FUNCTION_BLOCK FB_UML_SC
VAR
	// Transition condition
	bInitFinished				: BOOL;
	bUseXmlFormat				: BOOL;
	bAllInfoCopiedToFile		: BOOL;
	bSendToMasterFinished		: BOOL;
	bSendToClientFinished		: BOOL;
	
	// Counters
	nCounterInit				: INT;
	nCounterSaveInitSettings	: INT;
	nCounterClearXml			: INT;
	nCounterFillXml				: INT;
	nCounterSaveXml				: INT;
	nCounterClearText			: INT;
	nCounterFillText			: INT;
	nCounterSaveText			: INT;
	nCounterGetMasterID			: INT;
	nCounterGetClientID			: INT;
	nCounterSendToMaster		: INT;
	nCounterSendToClient		: INT;
	
	// Debugging
	bMasterFirst				: BOOL;
	bClientFirst				: BOOL;
END_VAR

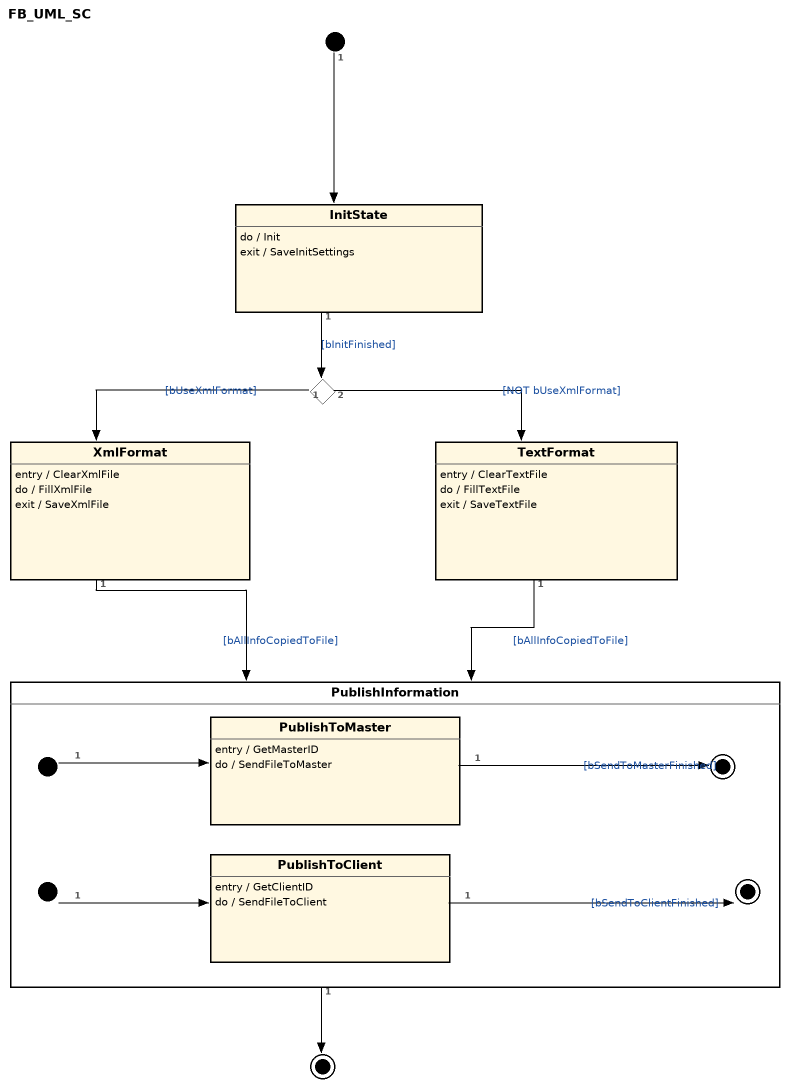
STATECHART FB_UML_SC  // abortable
    START StartState1
    STATE InitState
        do / Init
        exit / SaveInitSettings
    CHOICE ChoiceElement1
    STATE XmlFormat
        entry / ClearXmlFile
        do / FillXmlFile
        exit / SaveXmlFile
    STATE TextFormat
        entry / ClearTextFile
        do / FillTextFile
        exit / SaveTextFile
    COMPOSITE STATE PublishInformation
        REGION Region0 // priority 1
        START StartState2
        STATE PublishToMaster
            entry / GetMasterID
            do / SendFileToMaster
        END EndState2
        StartState2 -> PublishToMaster  // priority 1, on completion
        PublishToMaster -> EndState2 [bSendToMasterFinished] // priority 1
        REGION Region1 // priority 2
        START StartState3
        STATE PublishToClient
            entry / GetClientID
            do / SendFileToClient
        END EndState3
        StartState3 -> PublishToClient  // priority 1, on completion
        PublishToClient -> EndState3 [bSendToClientFinished] // priority 1
    END_STATE
    END EndState1
    StartState1 -> InitState  // priority 1, on completion
    InitState -> ChoiceElement1 [bInitFinished] // priority 1
    ChoiceElement1 -> XmlFormat [bUseXmlFormat] // priority 1
    ChoiceElement1 -> TextFormat [NOT bUseXmlFormat] // priority 2
    XmlFormat -> PublishInformation [bAllInfoCopiedToFile] // priority 1
    TextFormat -> PublishInformation [bAllInfoCopiedToFile] // priority 1
    PublishInformation -> EndState1  // priority 1, on completion
END_STATECHART

METHOD PROTECTED ClearTextFile
VAR_INPUT
END_VAR
nCounterClearText := nCounterClearText + 1;
END_METHOD

METHOD PROTECTED ClearXmlFile
VAR_INPUT
END_VAR
nCounterClearXml := nCounterClearXml + 1;
END_METHOD

METHOD PROTECTED FillTextFile
VAR_INPUT
END_VAR
nCounterFillText := nCounterFillText + 1;
END_METHOD

METHOD PROTECTED FillXmlFile
VAR_INPUT
END_VAR
nCounterFillXml := nCounterFillXml + 1;
END_METHOD

METHOD PROTECTED GetClientID
VAR_INPUT
END_VAR
nCounterGetClientID := nCounterGetClientID + 1;

IF NOT bMasterFirst THEN
	bClientFirst := TRUE;
END_IF
END_METHOD

METHOD PROTECTED GetMasterID
VAR_INPUT
END_VAR
nCounterGetMasterID := nCounterGetMasterID + 1;

IF NOT bClientFirst THEN
	bMasterFirst := TRUE;
END_IF
END_METHOD

METHOD PROTECTED Init
VAR_INPUT
END_VAR
nCounterInit := nCounterInit + 1;
END_METHOD

METHOD PROTECTED SaveInitSettings
VAR_INPUT
END_VAR
nCounterSaveInitSettings := nCounterSaveInitSettings + 1;

bInitFinished 			:= FALSE;
bAllInfoCopiedToFile 	:= FALSE;
bSendToClientFinished 	:= FALSE;
bSendToMasterFinished	:= FALSE;
bMasterFirst			:= FALSE;
bClientFirst			:= FALSE;
END_METHOD

METHOD PROTECTED SaveTextFile
VAR_INPUT
END_VAR
nCounterSaveText := nCounterSaveText + 1;
END_METHOD

METHOD PROTECTED SaveXmlFile
VAR_INPUT
END_VAR
nCounterSaveXml := nCounterSaveXml + 1;
END_METHOD

METHOD PROTECTED SendFileToClient
VAR_INPUT
END_VAR
nCounterSendToClient := nCounterSendToClient + 1;
END_METHOD

METHOD PROTECTED SendFileToMaster
VAR_INPUT
END_VAR
nCounterSendToMaster := nCounterSendToMaster + 1;
END_METHOD

END_FUNCTION_BLOCK

(* stored: Version 1.1.0.1, ProductVersion 3.1.4024.12
   POU FB_UML_SC: Id {94bc9ba2-99d4-44d6-a994-09cf55f5519b}, SpecialFunc None
   Method ClearTextFile: Id {eeadfa1a-8f3e-409c-821b-99021356a54f}
   Method ClearXmlFile: Id {f8f23fcf-54cf-4de2-a6bf-21ea7d0b73a5}
   Method FillTextFile: Id {8e04a295-480a-485c-95c5-43fbc530c30f}
   Method FillXmlFile: Id {414f740d-8f18-48da-80b3-7ea980956d61}
   Method GetClientID: Id {44e9e658-ee86-4494-b16a-b41b020447f1}
   Method GetMasterID: Id {7eaab2ed-ff02-4343-af44-fa07d4b58265}
   Method Init: Id {d0ad6e03-56a4-40f3-af43-3842eefeae86}
   Method SaveInitSettings: Id {a9fa5c00-a88c-49ee-a68d-e225192550e9}
   Method SaveTextFile: Id {219e5281-819e-448b-8b19-3e98bf2a2af0}
   Method SaveXmlFile: Id {03a23303-469c-4aa1-811c-347cee96a6ae}
   Method SendFileToClient: Id {f85a10a5-2d11-4ea8-a2ff-5eb2dc2ad2e9}
   Method SendFileToMaster: Id {2b74f887-17a5-4007-b86e-e2a7c00823a7} *)
